FUNCTION_BLOCK fbSimHSV
VAR_INPUT
	CmdOut : BOOL;
END_VAR
VAR_OUTPUT
	OpenSen : BOOL;
	CloseSen : BOOL;
END_VAR
VAR
	tOpenning : TIME := T#50MS;
	tonOpenning : TON;
	tClosing : TIME := T#50MS;
	tonClosing : TON;
END_VAR

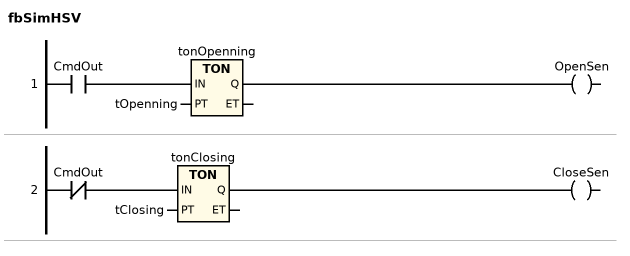
// NETWORK 1
tonOpenning(IN := CmdOut, PT := tOpenning); // TON
OpenSen := tonOpenning.Q;

// NETWORK 2
tonClosing(IN := NOT CmdOut, PT := tClosing); // TON
CloseSen := tonClosing.Q;

END_FUNCTION_BLOCK

(* stored: Version 1.1.0.1, ProductVersion 3.1.4022.17
   POU fbSimHSV: Id {0de70283-6cf1-43bb-b080-9757f558ac0b}, SpecialFunc None *)
